(* CoDeSys 2.3 library: ПЛК_ПЧВ_v2.lib *)
(* Libraries: Util.lib*11.12.18 13:38:51, STANDARD.LIB 4.10.05 11:14:46, IECSFC.LIB 13.4.06 15:51:28, SYSLIBTIME.LIB 20.2.06 12:31:16, SYSTASKINFO.LIB 20.2.06 12:31:38, ANALYZATION.LIB 5.10.99 09:05:06 *)

(* POU com_word_fb, ST *)
FUNCTION_BLOCK com_word_fb			(*ф.б. разбора коммандного слова*)
VAR_INPUT
	pre_task_num:BYTE:=1;					(*выбор номера предустановленного задания, доступные значения 1...4*)
	dc_stop:BOOL;							(*останов постоянным током*)
	slow_stop: BOOL;							(*останов выбегом*)
	fast_stop: BOOL;							(*быстрый останов*)
	start: BOOL;								(*пуск*)
	reverse: BOOL;							(*реверс*)
END_VAR
VAR
	bit_Low, bit_High:BOOL;					(*младший и старший биты выбора предустановленного задания*)
END_VAR
VAR_OUTPUT
	com_word:WORD;						(*регистр коммандного слова*)
END_VAR
(*приоритет выбора останова в случае одновремменной подачи нескольких сигналов *)
IF NOT(start) THEN										(*останов с замедлением*)
	dc_stop:=0;
	slow_stop:=0;
	fast_stop:=0;
ELSE														(*если нет останова с замедлением, то ...*)
	IF dc_stop THEN										(*останов постоянным током*)
		slow_stop:=0;
		fast_stop:=0;
	ELSE													(*если нет останова постоянным током, то ...*)
		IF slow_stop THEN								(*останов выбегом*)
			fast_stop:=0;
		END_IF											(*если нет останова выбегом, то смотрим состояние быстрого останова*)
	END_IF
END_IF

(*выбор номера предустановленного задания, для коммандного слова возможно задать только одно
из первых 4-х предустановленных заданий, предустановленное задание суммируется с основным заданием по интерфейсу*)
IF pre_task_num=1THEN
bit_Low:=0;
bit_High:=0;
ELSIF pre_task_num=2 THEN
bit_Low:=1;
bit_High:=0;
ELSIF pre_task_num=3 THEN
bit_Low:=0;
bit_High:=1;
ELSIF pre_task_num=4 THEN
bit_Low:=1;
bit_High:=1;
END_IF

(*разбор коммандного слова, подробное описание параметров в РПР и РПП на ПЧВ*)
com_word.0:=bit_Low;								(*выбор предустановленного задания, младший бит*)
com_word.1:=bit_High;								(*выбор предустановленноого задания, старший бит*)
com_word.2:=NOT(dc_stop);							(*нет торможения постоянным током*)
com_word.3:=NOT(slow_stop);						(*нет останова выбегом*)
com_word.4:=NOT(fast_stop);						(*нет быстрого останова*)
com_word.5:=1;										(*нет фиксации частоты*)
com_word.6:=start;									(*пуск*)
com_word.7:=0;										(*нет сброса*)
com_word.8:=0;										(*работа по заданию*)
com_word.9:=0;										(*изменение скорости 1*)
com_word.10:=1;										(*данные действительны*)
com_word.11:=0;										(*реле 1 выключено*)
com_word.12:=0;										(*не используется*)
com_word.13:=0;										(*не используется*)
com_word.14:=0;										(*набор 1*)
com_word.15:=reverse;								(*реверс*)
END_FUNCTION_BLOCK

(* POU stat_word_fb, ST *)
FUNCTION_BLOCK stat_word_fb			(*ф.б. разбора слова состояния*)
VAR_INPUT
	stat_word:WORD;							(*регистр слова состояния*)
END_VAR
VAR_OUTPUT
	ready_engine: BOOL;						(*готовность к управлению двигателя*)
	ready_drvive: BOOL;						(*готовность к управлению привода*)
	slow_stop_stat: BOOL;					(*останов выбегом, true - нет останова выбегом*)
	alarm: BOOL;								(*авария*)
	warning: BOOL;							(*предупреждение*)
	task_stat: BOOL;							(*выход на задание*)
	avt: BOOL;									(*режим работы, true - автоматический*)
	over_range: BOOL;						(*выход за частотный диапазон, true - в диапазоне*)
	work_stat: BOOL;							(*состояние, true - работа*)
	voltage: BOOL;							(*перенапряжение*)
	current: BOOL;							(*превышение предела по току*)
	heat: BOOL;								(*перегрев*)
END_VAR
(*разбор слова состояния привода, подробное описание параметров в РПР и РПП на ПЧВ*)
ready_engine:=stat_word.0;								(*готовность к управлению двигателя*)
ready_drvive:=stat_word.1;								(*готовность к управлению привода*)
slow_stop_stat:=stat_word.2;							(*останов выбегом*)
alarm:=stat_word.3;										(*авария*)
warning:=stat_word.7;									(*предупреждение*)
task_stat:=stat_word.8;									(*на задании/ не на задании*)
avt:=stat_word.9;											(*режим ручной/автоматический*)
over_range:=stat_word.10;								(* вне/в частотном диапазоне*)
work_stat:=stat_word.11;									(*останов/работа*)
voltage:=stat_word.13;									(*перенапряжение*)
current:=stat_word.14;									(*превышение предела по току*)
heat:=stat_word.15;										(*перегрев*)
END_FUNCTION_BLOCK

(* POU task_fb, ST *)
FUNCTION_BLOCK task_fb					(*ф.б. пересчета уставок задания*)
VAR_INPUT
	t_min: REAL;								(*минимальное задание, Гц*)
	t_max: REAL:=50;							(*максимальное задание, Гц*)
	task_value: REAL;							(*задание по интерфейсу RS485, %*)
	pre_task_value1: REAL;					(*предустановленное задание 1, %*)
	pre_task_value2: REAL;					(*предустановленное задание 2, %*)
	pre_task_value3: REAL;					(*предустановленное задание 3, %*)
	pre_task_value4: REAL;					(*предустановленное задание 4, %*)
	num_task: BYTE:=1;						(*номер предустановленного задания, доступные значения 1...8*)
	lim_h: REAL:=50;							(*верхний предел скорости вращения двигателя, Гц*)
	Idc_stop_val:WORD:=10;					(*ток торможения постоянным током, %*)
	rs_off: BOOL;								(*отключение источника задания 1, true - выключен, false - включен RS485, суммируется обычное задание и предустановленное*)
END_VAR
VAR_OUTPUT
	task_min: DWORD;						(*регистр минимального задания*)
	task_max: DWORD;						(*регистр максимального задания*)
	task: WORD;								(*регистр задания по интерфейсу RS485*)
	pre_task_value: WORD;					(*регистр предустановленного задания*)
	pre_task_num: WORD;					(*регистр номера предустановленного задания*)
	lim_high: WORD;							(*регистр верхнего предела скорости вращения двигателя*)
	Idc_stop:WORD;							(*регистр тока торможения постоянным током*)
	rs_out: WORD;							(*регистр отключения источника задания*)
END_VAR
VAR
	L_T: LIN_TRAFO;							(*ф.б. линейного преобразования значений из одного диапазона в другой, библиотека Util.lib*)
END_VAR
(*используем ф.б. линейного преобразования значений для приведения значения частоты в необходимый диапазон задания для ПЧВ*)
L_T(IN:=task_value, IN_MIN:=0, IN_MAX:=100, OUT_MIN:=0, OUT_MAX:=16384);
task:=REAL_TO_WORD(L_T.OUT);

(*установка минимального и максимального значений задания*)
task_min:=REAL_TO_DWORD(t_min*1000);
task_max:=REAL_TO_DWORD(t_max*1000);

(*выбор номера предустановленного задания и установка предустановленного задания*)
IF num_task=1 THEN
pre_task_num:=0;
pre_task_value:=REAL_TO_WORD(pre_task_value1*100);
ELSIF num_task=2 THEN
pre_task_num:=1;
pre_task_value:=REAL_TO_WORD(pre_task_value2*100);
ELSIF num_task=3 THEN
pre_task_num:=2;
pre_task_value:=REAL_TO_WORD(pre_task_value3*100);
ELSIF num_task=4 THEN
pre_task_num:=3;
pre_task_value:=REAL_TO_WORD(pre_task_value4*100);
ELSIF num_task=5 THEN
pre_task_num:=4;
END_IF

(*установка верхнего предела скорости вращения двигателя*)
lim_high:=REAL_TO_WORD(lim_h*10);

(*включение/отключение задания по интерфейсу*)
IF rs_off THEN
rs_out:=0;
ELSE
rs_out:=11;
END_IF

(*перевод значения тока торможения постоянным током*)
Idc_stop:=Idc_stop_val;
END_FUNCTION_BLOCK

(* POU value_fb, ST *)
FUNCTION_BLOCK value_fb					(*ф.б. определения значений мощности, напряжения, частоты и тока*)
VAR_INPUT
	P_:WORD;									(*регистр мощности*)
	U_:WORD;								(*регистр напряжения*)
	f_:WORD;									(*регситр частоты*)
	I_:WORD;									(*регистр тока*)
END_VAR
VAR_OUTPUT
	P: REAL;									(*мощность, кВт*)
	U: REAL;									(*напряжение, В*)
	f: REAL;									(*частота, Гц*)
	I: REAL;									(*ток, А*)
END_VAR
(*определение значений мощности, напряжения, частоты и тока*)
P:=WORD_TO_REAL(P_)/1000;							(*мощность, кВт*)
U:=WORD_TO_REAL(U_);								(*напряжение, В*)
f:=WORD_TO_REAL(f_)/10;								(*частота, Гц*)
I:=WORD_TO_REAL(I_)/100;								(*ток, А*)
END_FUNCTION_BLOCK
